INTERFACE I_SynchronousRpcHandler EXTENDS __SYSTEM.IQueryInterface

METHOD Handle
VAR_INPUT
	Parameters : I_Deserializer;
	Response : I_SynchronousRpcResponse;
END_VAR
END_METHOD

END_INTERFACE

(* stored: Version 1.1.0.1, ProductVersion 3.1.4026.13
   Itf I_SynchronousRpcHandler: Id {bd7246d2-6912-454e-8284-1058d0fb4690}
   Method Handle: Id {e6ba7fe5-059d-448d-ac0c-79caa69dc2e7} *)
